// TIA Portal V20 export
FUNCTION_BLOCK "LER_Recipe"   // FB213, LAD
// stored: Access Published, MemoryReserve 100, SetENOAutomatically false
   VAR_INPUT
      enable : Bool;
      applyBT : Bool;
   END_VAR
   VAR_IN_OUT
      parameterRecipeInterface : "HMI_IF_Parameter_LIstRecipe_Interface";
      parameterListSV : "HMI_IF_Parameter_ListRecipe_UDT";
      parameterListPV : "HMI_IF_Parameter_ListRecipe_UDT";
   END_VAR
   VAR_TEMP   // added for the SCL form of the ladder/FBD networks
      _w1 : Bool;
      _w2 : Bool;
   END_VAR
BEGIN

REGION Network 1: Recipe Chage
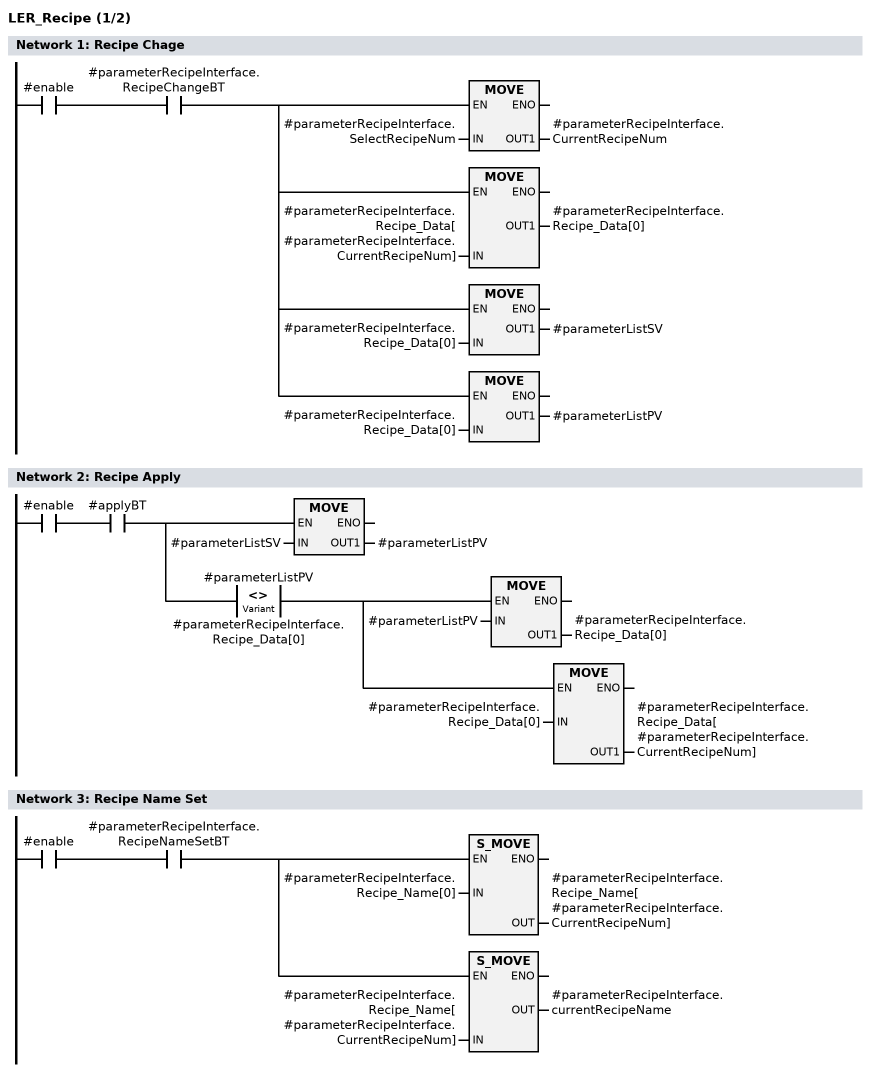
   RUNG wire#powerrail
      Contact( #enable )
      Contact( #parameterRecipeInterface.RecipeChangeBT )
      wire#w1
      { S7_GenerateENO := "TRUE" } Move(in := #parameterRecipeInterface.SelectRecipeNum, out1 => #parameterRecipeInterface.CurrentRecipeNum)
   END_RUNG
   RUNG wire#w1
      { S7_GenerateENO := "TRUE" } Move(in := #parameterRecipeInterface.Recipe_Data[#parameterRecipeInterface.CurrentRecipeNum], out1 => #parameterRecipeInterface.Recipe_Data[0])
   END_RUNG
   RUNG wire#w1
      { S7_GenerateENO := "TRUE" } Move(in := #parameterRecipeInterface.Recipe_Data[0], out1 => #parameterListSV)
   END_RUNG
   RUNG wire#w1
      { S7_GenerateENO := "TRUE" } Move(in := #parameterRecipeInterface.Recipe_Data[0], out1 => #parameterListPV)
   END_RUNG
   // the same network as SCL:
   IF #enable AND #parameterRecipeInterface.RecipeChangeBT THEN
       #parameterRecipeInterface.CurrentRecipeNum := #parameterRecipeInterface.SelectRecipeNum;
       #parameterRecipeInterface.Recipe_Data[0] := #parameterRecipeInterface.Recipe_Data[#parameterRecipeInterface.CurrentRecipeNum];
       #parameterListSV := #parameterRecipeInterface.Recipe_Data[0];
       #parameterListPV := #parameterRecipeInterface.Recipe_Data[0];
   END_IF;
END_REGION

REGION Network 2: Recipe Apply
   RUNG wire#powerrail
      Contact( #enable )
      Contact( #applyBT )
      wire#w1
      { S7_GenerateENO := "TRUE" } Move(in := #parameterListSV, out1 => #parameterListPV)
   END_RUNG
   RUNG wire#w1
      { S7_Templates := "SrcType := Variant" } NE_Contact(in1 := #parameterListPV, in2 := #parameterRecipeInterface.Recipe_Data[0])
      wire#w2
      { S7_GenerateENO := "TRUE" } Move(in := #parameterListPV, out1 => #parameterRecipeInterface.Recipe_Data[0])
   END_RUNG
   RUNG wire#w2
      { S7_GenerateENO := "TRUE" } Move(in := #parameterRecipeInterface.Recipe_Data[0], out1 => #parameterRecipeInterface.Recipe_Data[#parameterRecipeInterface.CurrentRecipeNum])
   END_RUNG
   // the same network as SCL:
   #_w1 := #enable AND #applyBT;
   IF #_w1 THEN #parameterListPV := #parameterListSV; END_IF;
   #_w2 := #_w1 AND (#parameterListPV <> #parameterRecipeInterface.Recipe_Data[0]);
   IF #_w2 THEN
       #parameterRecipeInterface.Recipe_Data[0] := #parameterListPV;
       #parameterRecipeInterface.Recipe_Data[#parameterRecipeInterface.CurrentRecipeNum] := #parameterRecipeInterface.Recipe_Data[0];
   END_IF;
END_REGION

REGION Network 3: Recipe Name Set
   RUNG wire#powerrail
      Contact( #enable )
      Contact( #parameterRecipeInterface.RecipeNameSetBT )
      wire#w1
      { S7_GenerateENO := "TRUE" } S_Move(in := #parameterRecipeInterface.Recipe_Name[0], out => #parameterRecipeInterface.Recipe_Name[#parameterRecipeInterface.CurrentRecipeNum])
   END_RUNG
   RUNG wire#w1
      { S7_GenerateENO := "TRUE" } S_Move(in := #parameterRecipeInterface.Recipe_Name[#parameterRecipeInterface.CurrentRecipeNum], out => #parameterRecipeInterface.currentRecipeName)
   END_RUNG
   // the same network as SCL:
   IF #enable AND #parameterRecipeInterface.RecipeNameSetBT THEN
       #parameterRecipeInterface.Recipe_Name[#parameterRecipeInterface.CurrentRecipeNum] := #parameterRecipeInterface.Recipe_Name[0];
       #parameterRecipeInterface.currentRecipeName := #parameterRecipeInterface.Recipe_Name[#parameterRecipeInterface.CurrentRecipeNum];
   END_IF;
END_REGION

REGION Network 4: Recipe Copy
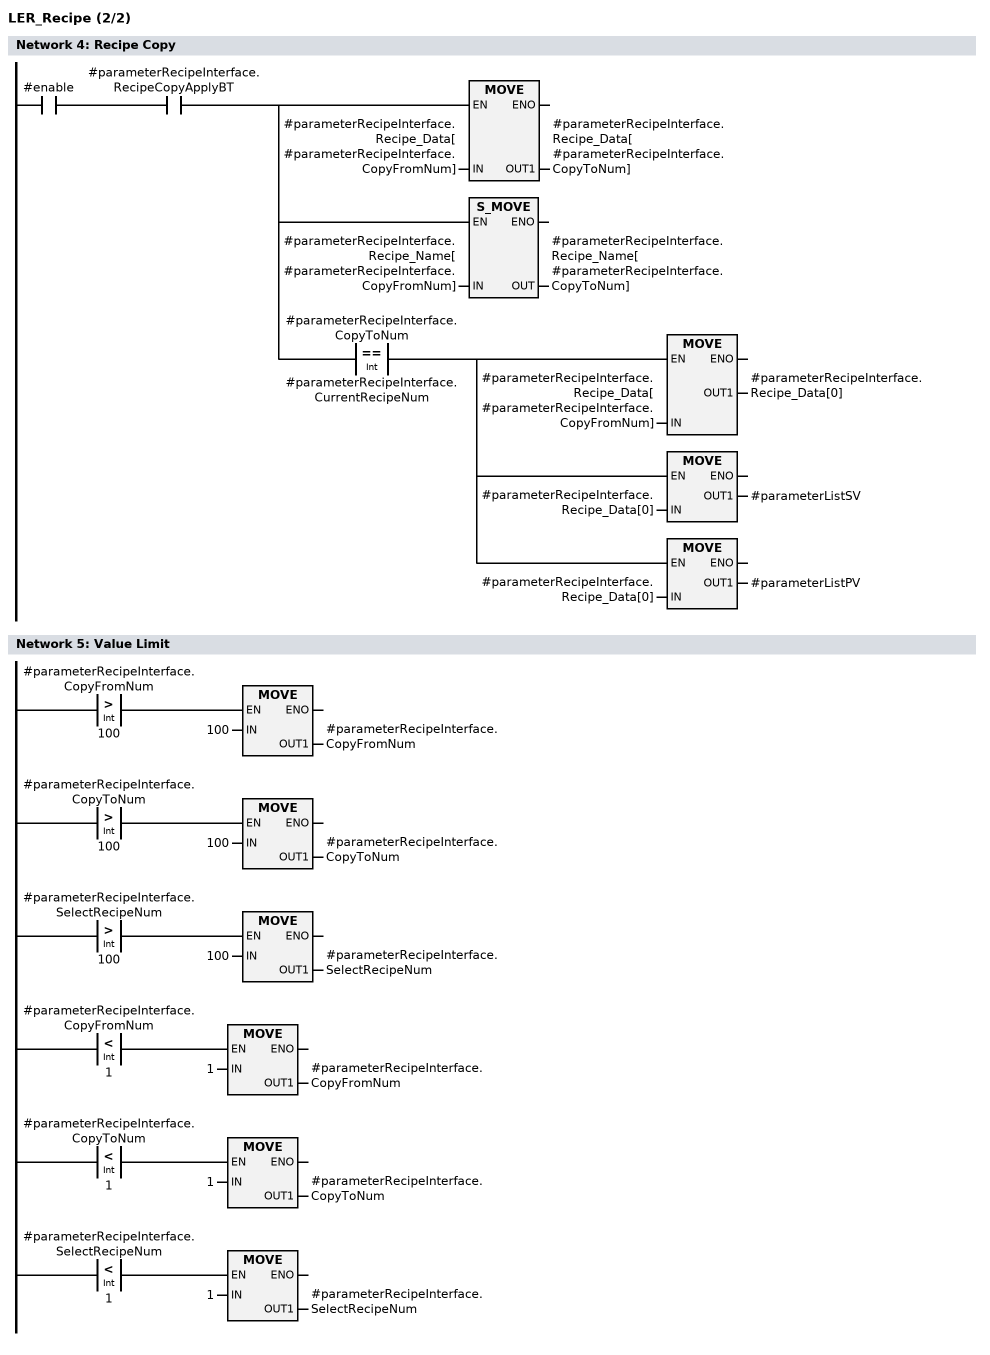
   RUNG wire#powerrail
      Contact( #enable )
      Contact( #parameterRecipeInterface.RecipeCopyApplyBT )
      wire#w1
      { S7_GenerateENO := "TRUE" } Move(in := #parameterRecipeInterface.Recipe_Data[#parameterRecipeInterface.CopyFromNum], out1 => #parameterRecipeInterface.Recipe_Data[#parameterRecipeInterface.CopyToNum])
   END_RUNG
   RUNG wire#w1
      { S7_GenerateENO := "TRUE" } S_Move(in := #parameterRecipeInterface.Recipe_Name[#parameterRecipeInterface.CopyFromNum], out => #parameterRecipeInterface.Recipe_Name[#parameterRecipeInterface.CopyToNum])
   END_RUNG
   RUNG wire#w1
      { S7_Templates := "SrcType := Int" } EQ_Contact(in1 := #parameterRecipeInterface.CopyToNum, in2 := #parameterRecipeInterface.CurrentRecipeNum)
      wire#w2
      { S7_GenerateENO := "TRUE" } Move(in := #parameterRecipeInterface.Recipe_Data[#parameterRecipeInterface.CopyFromNum], out1 => #parameterRecipeInterface.Recipe_Data[0])
   END_RUNG
   RUNG wire#w2
      { S7_GenerateENO := "TRUE" } Move(in := #parameterRecipeInterface.Recipe_Data[0], out1 => #parameterListSV)
   END_RUNG
   RUNG wire#w2
      { S7_GenerateENO := "TRUE" } Move(in := #parameterRecipeInterface.Recipe_Data[0], out1 => #parameterListPV)
   END_RUNG
   // the same network as SCL:
   #_w1 := #enable AND #parameterRecipeInterface.RecipeCopyApplyBT;
   IF #_w1 THEN
       #parameterRecipeInterface.Recipe_Data[#parameterRecipeInterface.CopyToNum] := #parameterRecipeInterface.Recipe_Data[#parameterRecipeInterface.CopyFromNum];
       #parameterRecipeInterface.Recipe_Name[#parameterRecipeInterface.CopyToNum] := #parameterRecipeInterface.Recipe_Name[#parameterRecipeInterface.CopyFromNum];
   END_IF;
   IF #_w1 AND (#parameterRecipeInterface.CopyToNum = #parameterRecipeInterface.CurrentRecipeNum) THEN
       #parameterRecipeInterface.Recipe_Data[0] := #parameterRecipeInterface.Recipe_Data[#parameterRecipeInterface.CopyFromNum];
       #parameterListSV := #parameterRecipeInterface.Recipe_Data[0];
       #parameterListPV := #parameterRecipeInterface.Recipe_Data[0];
   END_IF;
END_REGION

REGION Network 5: Value Limit
   RUNG wire#powerrail
      { S7_Templates := "SrcType := Int" } GT_Contact(in1 := #parameterRecipeInterface.CopyFromNum, in2 := 100)
      { S7_GenerateENO := "TRUE" } Move(in := 100, out1 => #parameterRecipeInterface.CopyFromNum)
   END_RUNG
   RUNG wire#powerrail
      { S7_Templates := "SrcType := Int" } GT_Contact(in1 := #parameterRecipeInterface.CopyToNum, in2 := 100)
      { S7_GenerateENO := "TRUE" } Move(in := 100, out1 => #parameterRecipeInterface.CopyToNum)
   END_RUNG
   RUNG wire#powerrail
      { S7_Templates := "SrcType := Int" } GT_Contact(in1 := #parameterRecipeInterface.SelectRecipeNum, in2 := 100)
      { S7_GenerateENO := "TRUE" } Move(in := 100, out1 => #parameterRecipeInterface.SelectRecipeNum)
   END_RUNG
   RUNG wire#powerrail
      { S7_Templates := "SrcType := Int" } LT_Contact(in1 := #parameterRecipeInterface.CopyFromNum, in2 := 1)
      { S7_GenerateENO := "TRUE" } Move(in := 1, out1 => #parameterRecipeInterface.CopyFromNum)
   END_RUNG
   RUNG wire#powerrail
      { S7_Templates := "SrcType := Int" } LT_Contact(in1 := #parameterRecipeInterface.CopyToNum, in2 := 1)
      { S7_GenerateENO := "TRUE" } Move(in := 1, out1 => #parameterRecipeInterface.CopyToNum)
   END_RUNG
   RUNG wire#powerrail
      { S7_Templates := "SrcType := Int" } LT_Contact(in1 := #parameterRecipeInterface.SelectRecipeNum, in2 := 1)
      { S7_GenerateENO := "TRUE" } Move(in := 1, out1 => #parameterRecipeInterface.SelectRecipeNum)
   END_RUNG
   // the same network as SCL:
   IF #parameterRecipeInterface.CopyFromNum > 100 THEN #parameterRecipeInterface.CopyFromNum := 100; END_IF;
   IF #parameterRecipeInterface.CopyToNum > 100 THEN #parameterRecipeInterface.CopyToNum := 100; END_IF;
   IF #parameterRecipeInterface.SelectRecipeNum > 100 THEN
       #parameterRecipeInterface.SelectRecipeNum := 100;
   END_IF;
   IF #parameterRecipeInterface.CopyFromNum < 1 THEN #parameterRecipeInterface.CopyFromNum := 1; END_IF;
   IF #parameterRecipeInterface.CopyToNum < 1 THEN #parameterRecipeInterface.CopyToNum := 1; END_IF;
   IF #parameterRecipeInterface.SelectRecipeNum < 1 THEN
       #parameterRecipeInterface.SelectRecipeNum := 1;
   END_IF;
END_REGION
END_FUNCTION_BLOCK
